// TIA Portal V15.1 export
// export: Created 2022-12-20T09:13:23.490063Z, ExportSetting None, DisplayName Totally Integrated Automation Portal, DisplayVersion V15.1 Update 1, DisplayName TIA Portal Openness, DisplayVersion V15.1, DisplayName SINAMICS Startdrive Advanced, DisplayVersion V15.1, DisplayName G130, G150, S120, S150, SINAMICS MV, S210, DisplayVersion V15.1, DisplayName G110M, G120, G120C, G120D, G120P, DisplayVersion V15.1, DisplayName STEP 7 Professional, DisplayVersion V15.1 Update 1, DisplayName STEP 7 Safety, DisplayVersion V15.1, DisplayName WinCC Professional, DisplayVersion V15.1 Update 1, DisplayName SIMATIC Visualization Architect, DisplayVersion V15.1
FUNCTION_BLOCK "SA01_TYPE_FB"   // FB904, FBD
TITLE = SA01_Type
{ S7_Optimized_Access := 'FALSE' }
// The block is used to control type movement throught the SA
// stored: AutoNumber false, SetENOAutomatically False
   VAR
      Simulation : "Type_Simulation_FB";   // Simulation
   END_VAR
BEGIN

REGION Network 1: *** Simulation ***
END_REGION

REGION Network 2: Type sim settings
   // Type sim settings
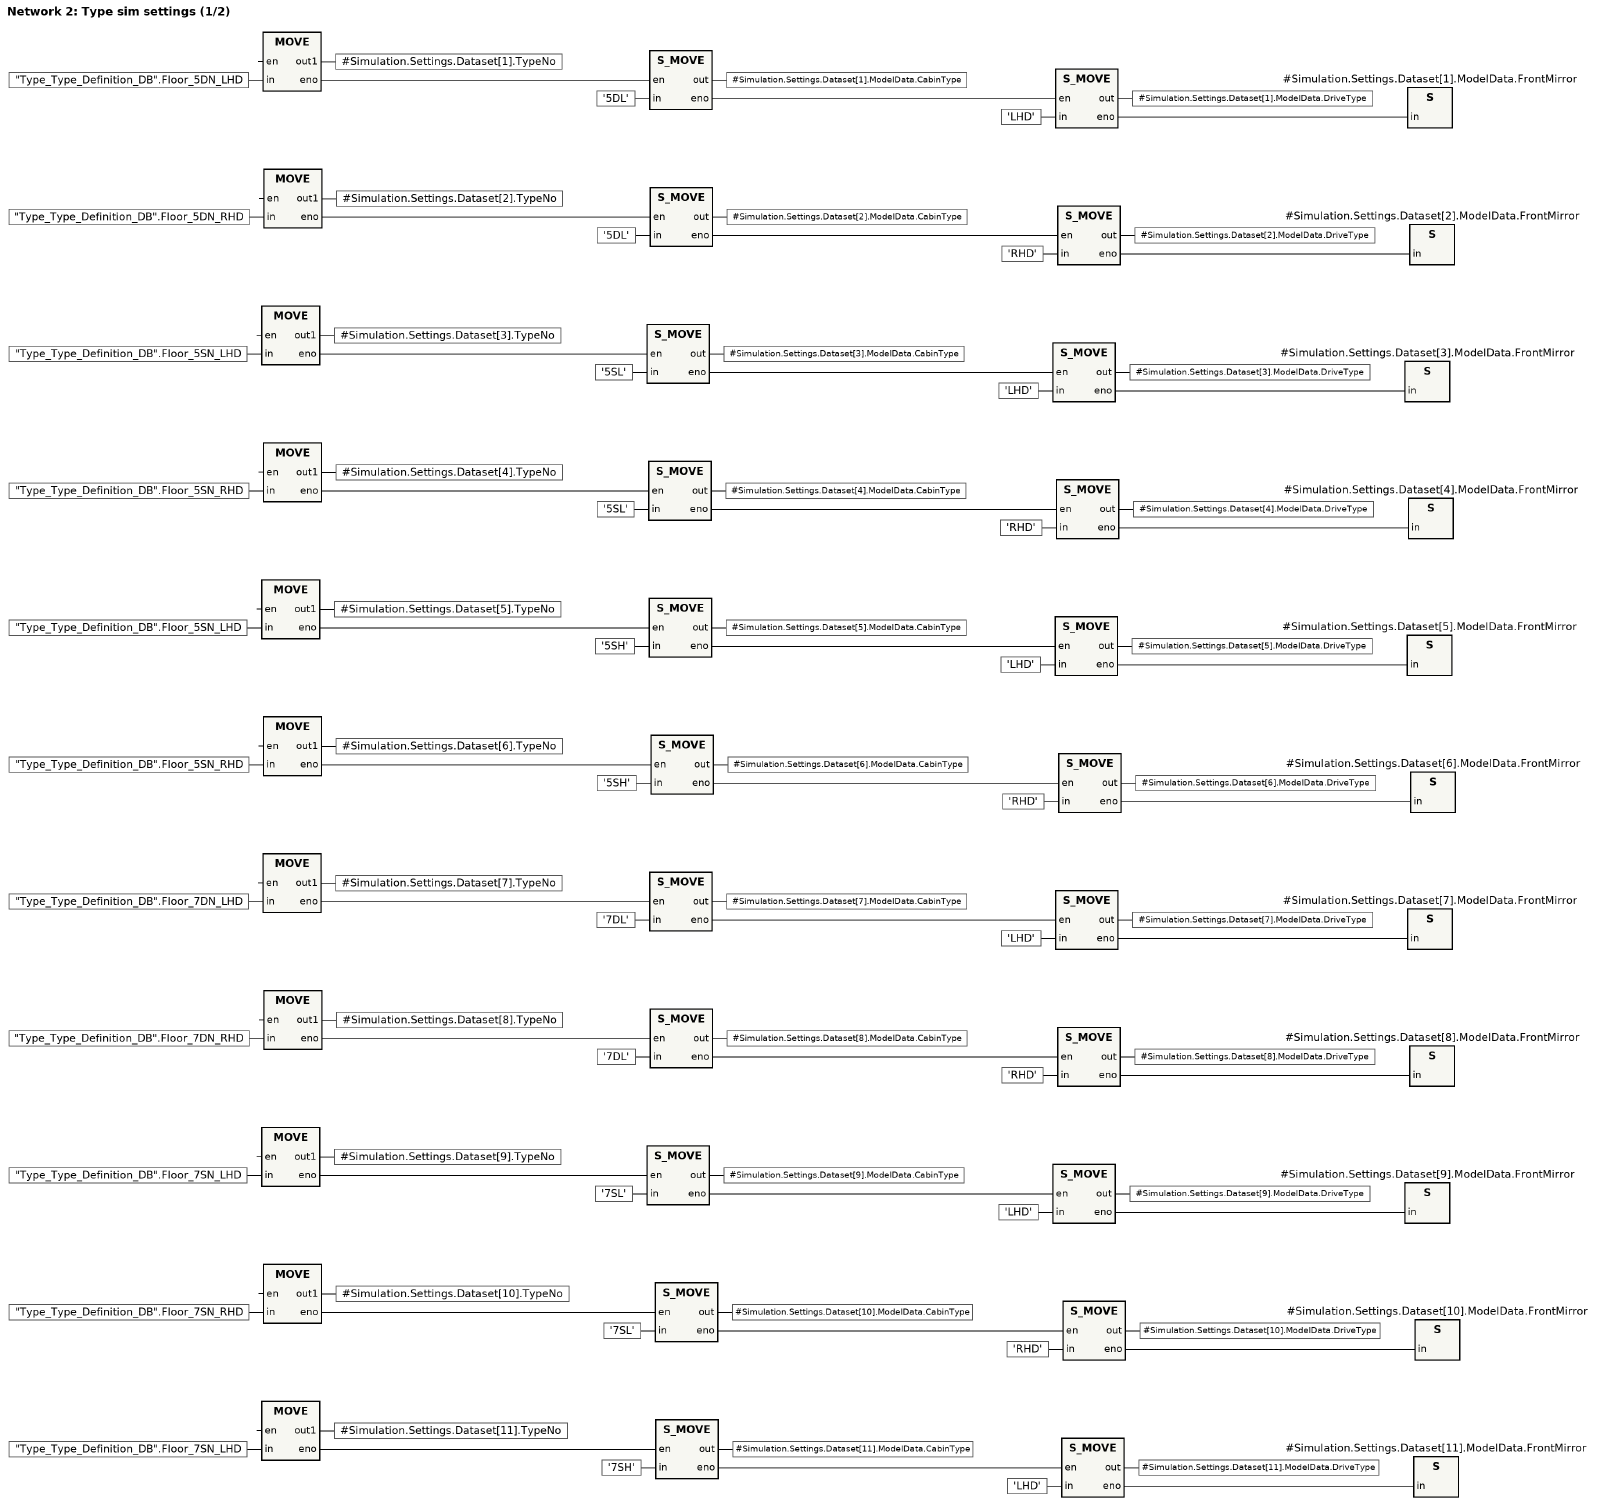
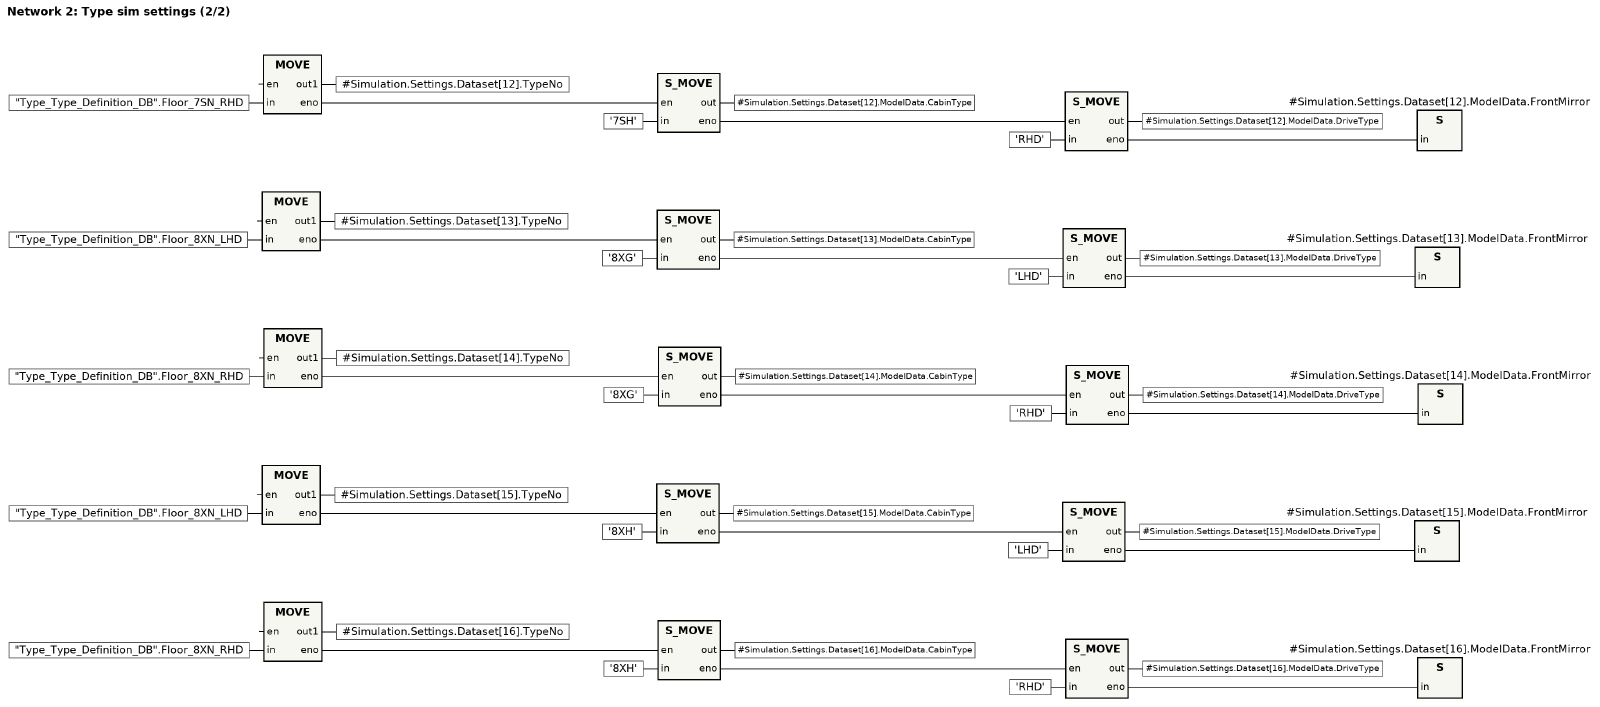
   #Simulation.Settings.Dataset[1].TypeNo := "Type_Type_Definition_DB".Floor_5DN_LHD;
   #Simulation.Settings.Dataset[1].ModelData.CabinType := '5DL';
   #Simulation.Settings.Dataset[1].ModelData.DriveType := 'LHD';
   #Simulation.Settings.Dataset[1].ModelData.FrontMirror := TRUE;
   #Simulation.Settings.Dataset[2].TypeNo := "Type_Type_Definition_DB".Floor_5DN_RHD;
   #Simulation.Settings.Dataset[2].ModelData.CabinType := '5DL';
   #Simulation.Settings.Dataset[2].ModelData.DriveType := 'RHD';
   #Simulation.Settings.Dataset[2].ModelData.FrontMirror := TRUE;
   #Simulation.Settings.Dataset[3].TypeNo := "Type_Type_Definition_DB".Floor_5SN_LHD;
   #Simulation.Settings.Dataset[3].ModelData.CabinType := '5SL';
   #Simulation.Settings.Dataset[3].ModelData.DriveType := 'LHD';
   #Simulation.Settings.Dataset[3].ModelData.FrontMirror := TRUE;
   #Simulation.Settings.Dataset[4].TypeNo := "Type_Type_Definition_DB".Floor_5SN_RHD;
   #Simulation.Settings.Dataset[4].ModelData.CabinType := '5SL';
   #Simulation.Settings.Dataset[4].ModelData.DriveType := 'RHD';
   #Simulation.Settings.Dataset[4].ModelData.FrontMirror := TRUE;
   #Simulation.Settings.Dataset[5].TypeNo := "Type_Type_Definition_DB".Floor_5SN_LHD;
   #Simulation.Settings.Dataset[5].ModelData.CabinType := '5SH';
   #Simulation.Settings.Dataset[5].ModelData.DriveType := 'LHD';
   #Simulation.Settings.Dataset[5].ModelData.FrontMirror := TRUE;
   #Simulation.Settings.Dataset[6].TypeNo := "Type_Type_Definition_DB".Floor_5SN_RHD;
   #Simulation.Settings.Dataset[6].ModelData.CabinType := '5SH';
   #Simulation.Settings.Dataset[6].ModelData.DriveType := 'RHD';
   #Simulation.Settings.Dataset[6].ModelData.FrontMirror := TRUE;
   #Simulation.Settings.Dataset[7].TypeNo := "Type_Type_Definition_DB".Floor_7DN_LHD;
   #Simulation.Settings.Dataset[7].ModelData.CabinType := '7DL';
   #Simulation.Settings.Dataset[7].ModelData.DriveType := 'LHD';
   #Simulation.Settings.Dataset[7].ModelData.FrontMirror := TRUE;
   #Simulation.Settings.Dataset[8].TypeNo := "Type_Type_Definition_DB".Floor_7DN_RHD;
   #Simulation.Settings.Dataset[8].ModelData.CabinType := '7DL';
   #Simulation.Settings.Dataset[8].ModelData.DriveType := 'RHD';
   #Simulation.Settings.Dataset[8].ModelData.FrontMirror := TRUE;
   #Simulation.Settings.Dataset[9].TypeNo := "Type_Type_Definition_DB".Floor_7SN_LHD;
   #Simulation.Settings.Dataset[9].ModelData.CabinType := '7SL';
   #Simulation.Settings.Dataset[9].ModelData.DriveType := 'LHD';
   #Simulation.Settings.Dataset[9].ModelData.FrontMirror := TRUE;
   #Simulation.Settings.Dataset[10].TypeNo := "Type_Type_Definition_DB".Floor_7SN_RHD;
   #Simulation.Settings.Dataset[10].ModelData.CabinType := '7SL';
   #Simulation.Settings.Dataset[10].ModelData.DriveType := 'RHD';
   #Simulation.Settings.Dataset[10].ModelData.FrontMirror := TRUE;
   #Simulation.Settings.Dataset[11].TypeNo := "Type_Type_Definition_DB".Floor_7SN_LHD;
   #Simulation.Settings.Dataset[11].ModelData.CabinType := '7SH';
   #Simulation.Settings.Dataset[11].ModelData.DriveType := 'LHD';
   #Simulation.Settings.Dataset[11].ModelData.FrontMirror := TRUE;
   #Simulation.Settings.Dataset[12].TypeNo := "Type_Type_Definition_DB".Floor_7SN_RHD;
   #Simulation.Settings.Dataset[12].ModelData.CabinType := '7SH';
   #Simulation.Settings.Dataset[12].ModelData.DriveType := 'RHD';
   #Simulation.Settings.Dataset[12].ModelData.FrontMirror := TRUE;
   #Simulation.Settings.Dataset[13].TypeNo := "Type_Type_Definition_DB".Floor_8XN_LHD;
   #Simulation.Settings.Dataset[13].ModelData.CabinType := '8XG';
   #Simulation.Settings.Dataset[13].ModelData.DriveType := 'LHD';
   #Simulation.Settings.Dataset[13].ModelData.FrontMirror := TRUE;
   #Simulation.Settings.Dataset[14].TypeNo := "Type_Type_Definition_DB".Floor_8XN_RHD;
   #Simulation.Settings.Dataset[14].ModelData.CabinType := '8XG';
   #Simulation.Settings.Dataset[14].ModelData.DriveType := 'RHD';
   #Simulation.Settings.Dataset[14].ModelData.FrontMirror := TRUE;
   #Simulation.Settings.Dataset[15].TypeNo := "Type_Type_Definition_DB".Floor_8XN_LHD;
   #Simulation.Settings.Dataset[15].ModelData.CabinType := '8XH';
   #Simulation.Settings.Dataset[15].ModelData.DriveType := 'LHD';
   #Simulation.Settings.Dataset[15].ModelData.FrontMirror := TRUE;
   #Simulation.Settings.Dataset[16].TypeNo := "Type_Type_Definition_DB".Floor_8XN_RHD;
   #Simulation.Settings.Dataset[16].ModelData.CabinType := '8XH';
   #Simulation.Settings.Dataset[16].ModelData.DriveType := 'RHD';
   #Simulation.Settings.Dataset[16].ModelData.FrontMirror := TRUE;
END_REGION

REGION Network 3: Type sim logic
   // Type sim logic
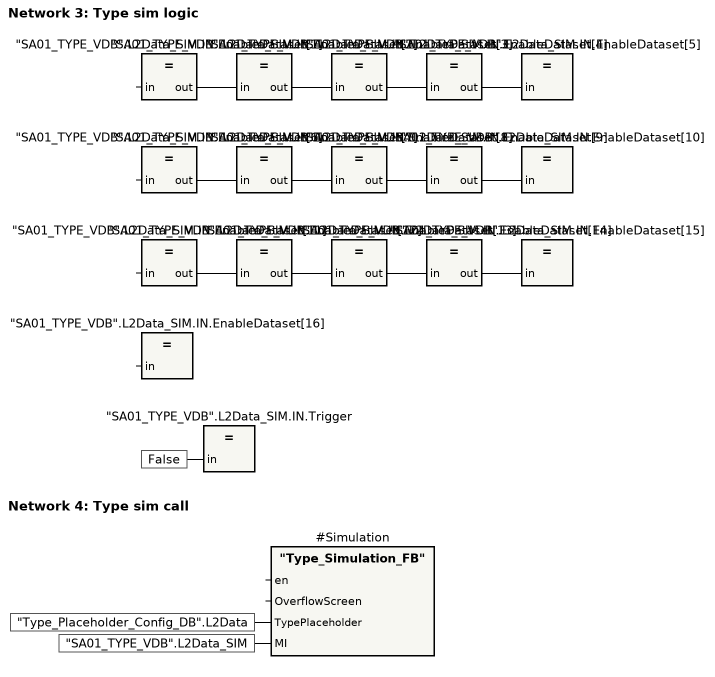
   "SA01_TYPE_VDB".L2Data_SIM.IN.EnableDataset[1] := TRUE;
   "SA01_TYPE_VDB".L2Data_SIM.IN.EnableDataset[2] := TRUE;
   "SA01_TYPE_VDB".L2Data_SIM.IN.EnableDataset[3] := TRUE;
   "SA01_TYPE_VDB".L2Data_SIM.IN.EnableDataset[4] := TRUE;
   "SA01_TYPE_VDB".L2Data_SIM.IN.EnableDataset[5] := TRUE;
   "SA01_TYPE_VDB".L2Data_SIM.IN.EnableDataset[6] := TRUE;
   "SA01_TYPE_VDB".L2Data_SIM.IN.EnableDataset[7] := TRUE;
   "SA01_TYPE_VDB".L2Data_SIM.IN.EnableDataset[8] := TRUE;
   "SA01_TYPE_VDB".L2Data_SIM.IN.EnableDataset[9] := TRUE;
   "SA01_TYPE_VDB".L2Data_SIM.IN.EnableDataset[10] := TRUE;
   "SA01_TYPE_VDB".L2Data_SIM.IN.EnableDataset[11] := TRUE;
   "SA01_TYPE_VDB".L2Data_SIM.IN.EnableDataset[12] := TRUE;
   "SA01_TYPE_VDB".L2Data_SIM.IN.EnableDataset[13] := TRUE;
   "SA01_TYPE_VDB".L2Data_SIM.IN.EnableDataset[14] := TRUE;
   "SA01_TYPE_VDB".L2Data_SIM.IN.EnableDataset[15] := TRUE;
   "SA01_TYPE_VDB".L2Data_SIM.IN.EnableDataset[16] := TRUE;
   "SA01_TYPE_VDB".L2Data_SIM.IN.Trigger := False;
END_REGION

REGION Network 4: Type sim call
   // Type sim call
   #Simulation(TypePlaceholder := "Type_Placeholder_Config_DB".L2Data, MI := "SA01_TYPE_VDB".L2Data_SIM);   // "Type_Simulation_FB"
END_REGION
END_FUNCTION_BLOCK
